TYPE ST_CompensationSummary :
STRUCT
    nTotalActiveCapacitors : INT;           // Toplam aktif kondansatör sayısı
    rTotalActivePower : REAL;               // Toplam aktif güç (kVAr)
    nActiveGroupCount : INT;                // Aktif grup sayısı
END_STRUCT
END_TYPE

(* stored: Version 1.1.0.1, ProductVersion 3.1.4024.15
   DUT ST_CompensationSummary: Id {da015f38-03cc-4a8c-925f-84f521aa7712} *)
